// TIA Portal project "PID学习" (V16)

(* hardware
DEVICE "S7-1200 station_1"  S7-1200 Station
   slot 0: "Rack_0"  S7-1200 Rack  Rack  V1.0
   slot 1: "PLC_1"  CPU 1214C DC/DC/Rly  6ES7 214-1HG40-0XB0  V4.4
   slot 2: "AI 4x13BIT/AQ 2x14BIT_1"  6ES7 234-4HE32-0XB0  V2.1
*)

// ===== PLC "PLC_1"  CPU 1214C DC/DC/Rly =====

VAR_GLOBAL   // PLC tag table "默认变量表"
   "Tag_1" AT %IW96 : Int;
   "Tag_2" AT %MW5 : Word;
   "启动PID" AT %M0.4 : Bool;
   "控制进水阀" AT %MD60 : DWord;
   "Tag_3" AT %QD30 : Real;
   "Tag_4" AT %QD60 : Real;
   "Tag_5" AT %Q2.3 : Bool;
   "System_Byte" AT %MB1 : Byte;
   "FirstScan" AT %M1.0 : Bool;
   "DiagStatusUpdate" AT %M1.1 : Bool;
   "AlwaysTRUE" AT %M1.2 : Bool;
   "AlwaysFALSE" AT %M1.3 : Bool;
   "Clock_Byte" AT %MB5 : Byte;
   "Clock_10Hz" AT %M5.0 : Bool;
   "Clock_5Hz" AT %M5.1 : Bool;
   "Clock_2.5Hz" AT %M5.2 : Bool;
   "Clock_2Hz" AT %M5.3 : Bool;
   "Clock_1.25Hz" AT %M5.4 : Bool;
   "Clock_1Hz" AT %M5.5 : Bool;
   "Clock_0.625Hz" AT %M5.6 : Bool;
   "Clock_0.5Hz" AT %M5.7 : Bool;
END_VAR

VAR_GLOBAL   // PLC tag table "io表"
   "启动开关" AT %I2.0 : Bool;
   "复位开关" AT %I2.1 : Bool;
   "停止开关" AT %I2.2 : Bool;
   "FACTORY I/O (Running)" AT %I2.3 : Bool;
   "启动指示灯" AT %Q2.0 : Bool;
   "复位指示灯" AT %Q2.1 : Bool;
   "停止指示灯" AT %Q2.2 : Bool;
   "定位点(1)" AT %ID38 : Real;
   "流量计" AT %ID34 : Real;
   "液位计" AT %ID30 : Real;
   "进水阀" AT %QD40 : Real;
   "排出阀" AT %QD44 : Real;
   "流液显示屏" AT %QD48 : DInt;
   "流量显示屏" AT %QD52 : DInt;
END_VAR

VAR_GLOBAL   // PLC tag table "变量表_1"
   "开启进水阀" AT %M0.0 : Bool;
   "温度转换" AT %MD10 : Real;
   "实际温度" AT %MD100 : Real;
   "流量转换" AT %MD14 : Real;
   "实际流量" AT %MD104 : Real;
   "中间变量1" AT %M0.1 : Bool;
   "开启排水阀" AT %M0.2 : Bool;
   "中间变量2" AT %M0.3 : Bool;
   "中间变量3" AT %M0.5 : Bool;
   "中间变量4" AT %M0.6 : Bool;
   "中间转换1" AT %MD30 : DInt;
   "中间转换2" AT %MD34 : DInt;
END_VAR

DATA_BLOCK "液位变量"   // DB2
{ S7_Optimized_Access := 'TRUE' }
VERSION : 0.1
   VAR
      PID设定值 : Real := 1500.0;
      过程值1 : Real;
      过程值2 : Real;
      过程值3 : Real;
      过程值4 : Real;
      过程值5 : Real;
      反馈值1 : Real;
      排水阀 : Real := 4.0;
      PID输出值 : Real := 100.0;
      pid的mode : Int;
      "Q2.0_P" : Bool;
      "Q2.1_N" : Bool;
      "Q2.3" : Bool;
      ModeActivate : Bool;
      ModeActivate_1 : Bool;
      Reset : Bool;
      State : Int;
      Error : Bool;
      ErrorBits : DInt;
   END_VAR
BEGIN
END_DATA_BLOCK

FUNCTION "模拟量" : Void   // FC1, LAD
{ S7_Optimized_Access := 'TRUE' }
VERSION : 0.1
BEGIN

REGION Network 1: 设定PID的设定值
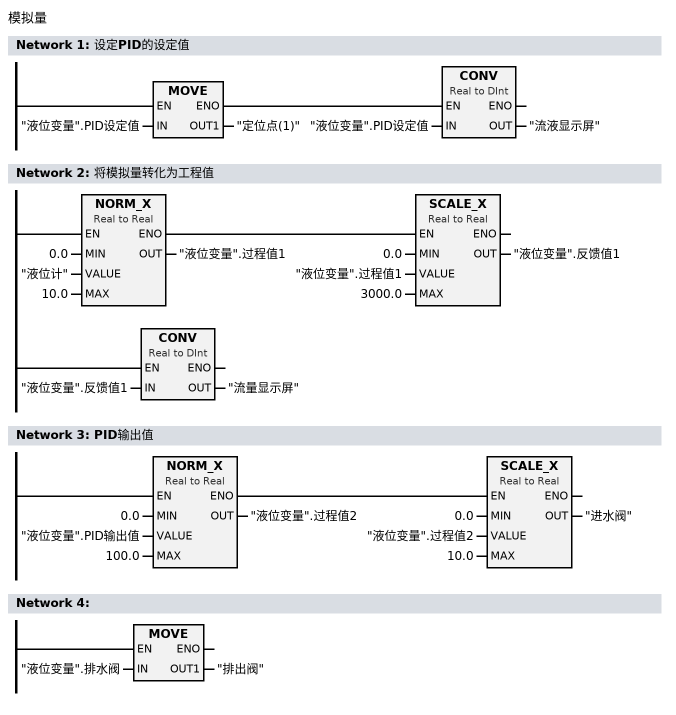
   RUNG wire#powerrail
      Move(in := "液位变量".PID设定值, out1 => "定位点(1)")
      { S7_Templates := "[SrcType := Real, DestType := DInt]" } Convert(in := "液位变量".PID设定值, out => "流液显示屏")
   END_RUNG
   // the same network as SCL:
   "定位点(1)" := "液位变量".PID设定值;
   "流液显示屏" := REAL_TO_DINT("液位变量".PID设定值);
END_REGION

REGION Network 2: 将模拟量转化为工程值
   RUNG wire#powerrail
      { S7_Templates := "[SrcType := Real, DestType := Real]" } Normalize(min := 0.0, value := "液位计", max := 10.0, out => "液位变量".过程值1)
      { S7_Templates := "[SrcType := Real, DestType := Real]" } Scale(min := 0.0, value := "液位变量".过程值1, max := 3000.0, out => "液位变量".反馈值1)
   END_RUNG
   RUNG wire#powerrail
      { S7_Templates := "[SrcType := Real, DestType := DInt]" } Convert(in := "液位变量".反馈值1, out => "流量显示屏")
   END_RUNG
   // the same network as SCL:
   "液位变量".过程值1 := NORM_X(MIN := 0.0, VALUE := "液位计", MAX := 10.0);
   "液位变量".反馈值1 := SCALE_X(MIN := 0.0, VALUE := "液位变量".过程值1, MAX := 3000.0);
   "流量显示屏" := REAL_TO_DINT("液位变量".反馈值1);
END_REGION

REGION Network 3: PID输出值
   RUNG wire#powerrail
      { S7_Templates := "[SrcType := Real, DestType := Real]" } Normalize(min := 0.0, value := "液位变量".PID输出值, max := 100.0, out => "液位变量".过程值2)
      { S7_Templates := "[SrcType := Real, DestType := Real]" } Scale(min := 0.0, value := "液位变量".过程值2, max := 10.0, out => "进水阀")
   END_RUNG
   // the same network as SCL:
   "液位变量".过程值2 := NORM_X(MIN := 0.0, VALUE := "液位变量".PID输出值, MAX := 100.0);
   "进水阀" := SCALE_X(MIN := 0.0, VALUE := "液位变量".过程值2, MAX := 10.0);
END_REGION

REGION Network 4
   RUNG wire#powerrail
      Move(in := "液位变量".排水阀, out1 => "排出阀")
   END_RUNG
   // the same network as SCL:
   "排出阀" := "液位变量".排水阀;
END_REGION
END_FUNCTION

FUNCTION "液位启停" : Void   // FC2, LAD
{ S7_Optimized_Access := 'TRUE' }
VERSION : 0.1
BEGIN

REGION Network 1
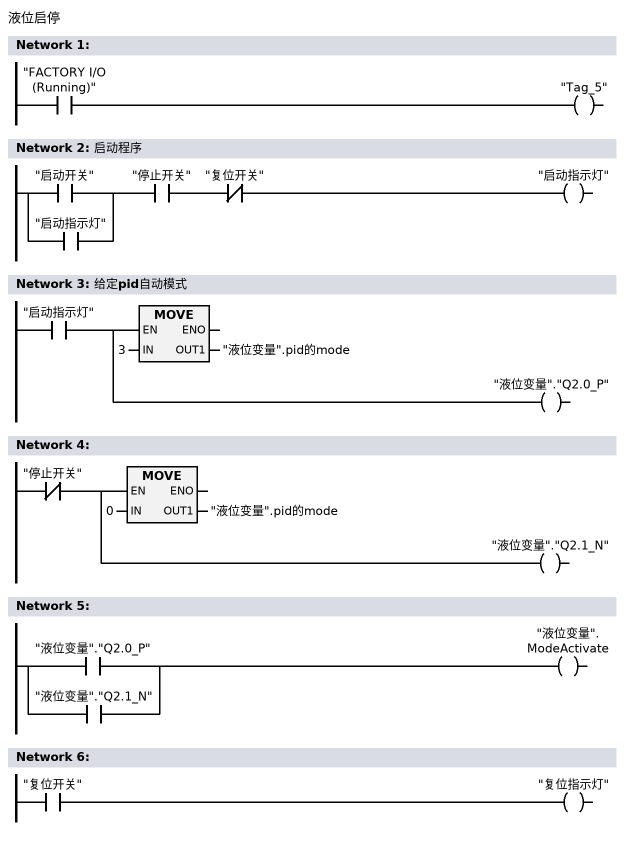
   RUNG wire#powerrail
      Contact( "FACTORY I/O (Running)" )
      Coil( "Tag_5" )
   END_RUNG
   // the same network as SCL:
   "Tag_5" := "FACTORY I/O (Running)";
END_REGION

REGION Network 2: 启动程序
   RUNG wire#powerrail
      Contact( "启动开关" )
      wire#w1
      Contact( "停止开关" )
      I_Contact( "复位开关" )
      Coil( "启动指示灯" )
   END_RUNG
   RUNG wire#powerrail
      Contact( "启动指示灯" )
   END_RUNG wire#w1
   // the same network as SCL:
   "启动指示灯" := ("启动开关" OR "启动指示灯") AND "停止开关" AND NOT "复位开关";
END_REGION

REGION Network 3: 给定pid自动模式
   RUNG wire#powerrail
      Contact( "启动指示灯" )
      wire#w1
      Move(in := 3, out1 => "液位变量".pid的mode)
   END_RUNG
   RUNG wire#w1
      Coil( "液位变量"."Q2.0_P" )
   END_RUNG
   // the same network as SCL:
   IF "启动指示灯" THEN "液位变量".pid的mode := 3; END_IF;
   "液位变量"."Q2.0_P" := "启动指示灯";
END_REGION

REGION Network 4
   RUNG wire#powerrail
      I_Contact( "停止开关" )
      wire#w1
      Move(in := 0, out1 => "液位变量".pid的mode)
   END_RUNG
   RUNG wire#w1
      Coil( "液位变量"."Q2.1_N" )
   END_RUNG
   // the same network as SCL:
   IF NOT "停止开关" THEN "液位变量".pid的mode := 0; END_IF;
   "液位变量"."Q2.1_N" := NOT "停止开关";
END_REGION

REGION Network 5
   RUNG wire#powerrail
      Contact( "液位变量"."Q2.0_P" )
      wire#w1
      Coil( "液位变量".ModeActivate )
   END_RUNG
   RUNG wire#powerrail
      Contact( "液位变量"."Q2.1_N" )
   END_RUNG wire#w1
   // the same network as SCL:
   "液位变量".ModeActivate := "液位变量"."Q2.0_P" OR "液位变量"."Q2.1_N";
END_REGION

REGION Network 6
   RUNG wire#powerrail
      Contact( "复位开关" )
      Coil( "复位指示灯" )
   END_RUNG
   // the same network as SCL:
   "复位指示灯" := "复位开关";
END_REGION
END_FUNCTION

FUNCTION "液位控制" : Void   // FC3, LAD
{ S7_Optimized_Access := 'TRUE' }
VERSION : 0.1
   VAR_TEMP   // added for the SCL form of the ladder/FBD networks
      _w1 : Bool;
   END_VAR
BEGIN

REGION Network 1
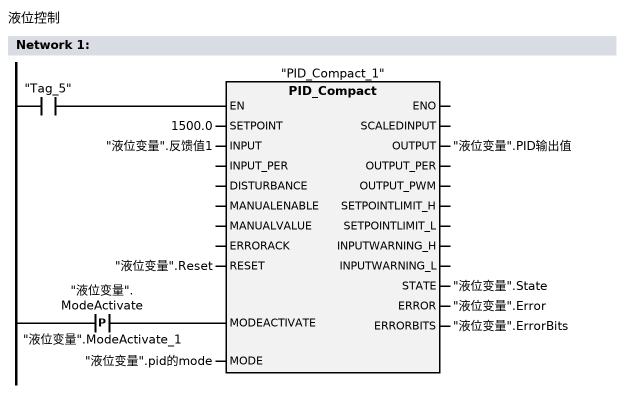
   #_w1 := "液位变量".ModeActivate AND NOT "液位变量".ModeActivate_1;   // rising edge of "液位变量".ModeActivate
   "液位变量".ModeActivate_1 := "液位变量".ModeActivate;
   IF "Tag_5" THEN
       "PID_Compact_1"(Setpoint := 1500.0,   // PID_Compact
                       Input := "液位变量".反馈值1,
                       Reset := "液位变量".Reset,
                       ModeActivate := #_w1,
                       Mode := "液位变量".pid的mode,
                       Output => "液位变量".PID输出值,
                       State => "液位变量".State,
                       Error => "液位变量".Error,
                       ErrorBits => "液位变量".ErrorBits);
   END_IF;
END_REGION
END_FUNCTION

FUNCTION "MHJ-PLC-Lab-Function-S71200" : Void   // FC9000, SCL
{ S7_Optimized_Access := 'TRUE' }
VERSION : 0.1
   VAR_TEMP
      rdTimeReturn : Int;
      outputTime : DTL;
      SyncVal : Byte;
      forVal : Int;
      forVal_2 : Int;
      Value : Byte;
   END_VAR
   VAR CONSTANT
      CompVal : Byte := 16#34;
      Value_01 : Byte := 16#11;
      Value_01_DW : DWord := 16#A165_D992;
      Value_02_DW : DWord := 16#58BE_4401;
   END_VAR
BEGIN

   #Value:=PEEK(area := 16#82,
        dbNumber := 0,
        byteOffset := 511);
   #Value := #Value + 1;

   POKE(area := 16#82,
        dbNumber := 0,
        byteOffset := 511,
        value := #Value);

   POKE(area:=16#81,
        dbNumber:=0,
        byteOffset:=1016,
        value:=#Value_01_DW);
   POKE(area := 16#81,
        dbNumber := 0,
        byteOffset := 1020,
        value := #Value_02_DW);

   POKE(area := 16#81,
        dbNumber := 0,
        byteOffset := 511,
        value := B#16#00);

   FOR #forVal := 0 TO 120 DO
       FOR #forVal_2:=0 TO 10 DO
           #rdTimeReturn:=RD_SYS_T(#outputTime);
           #rdTimeReturn := WR_SYS_T(#outputTime);
           #rdTimeReturn := RD_SYS_T(#outputTime);
           #rdTimeReturn := WR_SYS_T(#outputTime);
       END_FOR;
       #SyncVal:= PEEK(area := 16#81,
                      dbNumber := 0,
                      byteOffset := 511);
       IF #SyncVal = #CompVal THEN
          GOTO M_1;
       END_IF;
   END_FOR;
   RETURN;

   M_1:
   POKE(area := 16#81,
        dbNumber := 0,
        byteOffset := 511,
        value := B#16#0);
END_FUNCTION

ORGANIZATION_BLOCK "Main"   // OB1, LAD, ProgramCycle
TITLE = "Main Program Sweep (Cycle)"
{ S7_Optimized_Access := 'TRUE' }
VERSION : 0.1
   VAR_INPUT
      Initial_Call : Bool;   // Initial call of this OB
      Remanence : Bool;   // =True, if remanent data are available
   END_VAR
BEGIN

REGION Network 1
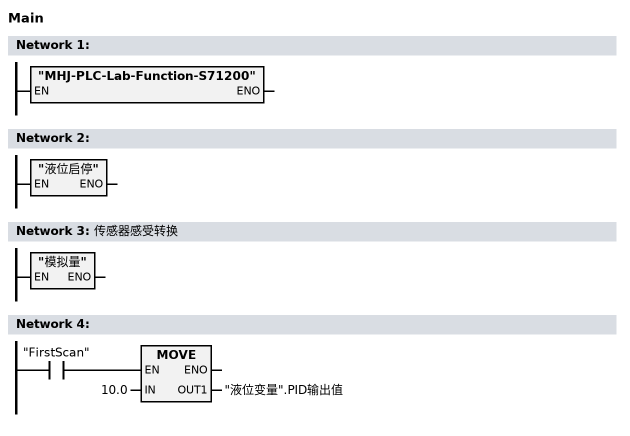
   RUNG wire#powerrail
      "MHJ-PLC-Lab-Function-S71200"()
   END_RUNG
   // the same network as SCL:
   "MHJ-PLC-Lab-Function-S71200"();
END_REGION

REGION Network 2
   RUNG wire#powerrail
      "液位启停"()
   END_RUNG
   // the same network as SCL:
   "液位启停"();
END_REGION

REGION Network 3: 传感器感受转换
   RUNG wire#powerrail
      "模拟量"()
   END_RUNG
   // the same network as SCL:
   "模拟量"();
END_REGION

REGION Network 4
   RUNG wire#powerrail
      Contact( "FirstScan" )
      Move(in := 10.0, out1 => "液位变量".PID输出值)
   END_RUNG
   // the same network as SCL:
   IF "FirstScan" THEN "液位变量".PID输出值 := 10.0; END_IF;
END_REGION
END_ORGANIZATION_BLOCK

ORGANIZATION_BLOCK "循环"   // OB30, LAD, CyclicInterrupt
{ S7_Optimized_Access := 'TRUE' }
VERSION : 0.1
   VAR_INPUT
      Initial_Call : Bool;   // Initial call of this OB
      Event_Count : Int;   // Events discarded
   END_VAR
BEGIN

REGION Network 1
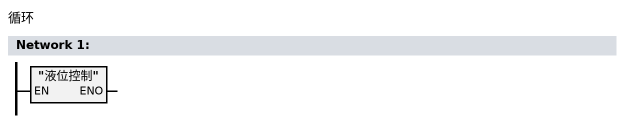
   RUNG wire#powerrail
      "液位控制"()
   END_RUNG
   // the same network as SCL:
   "液位控制"();
END_REGION
END_ORGANIZATION_BLOCK